Staubli VAL3: Digtal2Analog.pgx

public program Digtal2Analog()
  local num l_nIndexX
  local num l_nIndexY
  local num l_nNum
  local string l_sIOName
begin

  //数字量转换为模拟量

  //  for l_nIndexY=0 to 4
  //    l_nNum=0
  //    for l_nIndexX =0 to 15
  //      call IOName(67+l_nIndexX+l_nIndexY*16,l_sIOName)
  //      if (67+l_nIndexX+l_nIndexY*16)<135
  //        l_nNum=l_nNum+sel(dDio[l_sIOName]==true,1,0)*power(2,l_nIndexX)
  //      endIf
  //    endFor
  //    call IOName(159+l_nIndexY,l_sIOName)
  //    aioSet(aAio[l_sIOName],l_nNum)
  //  //  delay(0)
  //  endFor
  //


  call Digtal2AnalogS(0)
  call Digtal2AnalogS(1)
  call Digtal2AnalogS(2)
  call Digtal2AnalogS(3)
  call Digtal2AnalogS(4)

end
